FUNCTION_BLOCK Test_TimeAsString_24HourFormat EXTENDS TUnitTestBase
VAR
    TimeStruct : TIMESTRUCT := (wHour := 22, wMinute := 20, wSecond := 18);
END_VAR

Assertion.AssertEquals_STRING(
    Expected := '22:20:18',
    Actual   := F_TimeAsString(TimeStruct),
    ObjectName := _TestName,
    VariableName  := 'F_TimeAsString(TimeStruct)');


Test_Finished();

END_FUNCTION_BLOCK

(* stored: Version 1.1.0.1, ProductVersion 3.1.4024.3
   POU Test_TimeAsString_24HourFormat: Id {f81aab76-2a34-01f9-2fb5-1c273e9923eb}, SpecialFunc None *)
